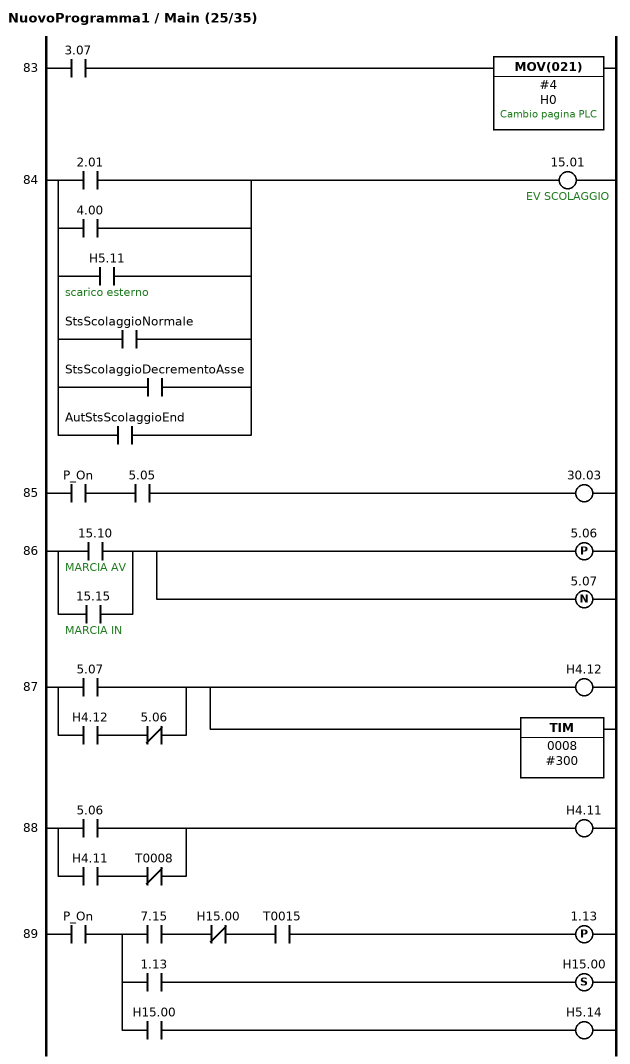
; [picture p24: NuovoProgramma1 / Main, rungs 83-89]
; rung 83
LD 3.07
MOV(021) #4 H0  ; Cambio pagina PLC
; rung 84
LD 2.01
OR 4.00
OR H5.11  ; scarico esterno
OR StsScolaggioNormale
OR StsScolaggioDecrementoAsse
OR AutStsScolaggioEnd
OUT 15.01  ; EV SCOLAGGIO
; rung 85
LD P_On
AND 5.05
OUT 30.03
; rung 86
LD 15.10  ; MARCIA AV
OR 15.15  ; MARCIA IN
DIFU(013) 5.06
DIFD(014) 5.07
; rung 87
LD 5.07
LD H4.12
ANDNOT 5.06
ORLD
OUT H4.12
TIM 0008 #300
; rung 88
LD 5.06
LD H4.11
ANDNOT T0008
ORLD
OUT H4.11
; rung 89
LD P_On
OUT TR0
AND 7.15
ANDNOT H15.00
AND T0015
DIFU(013) 1.13
LD TR0
AND 1.13
SET H15.00
LD TR0
AND H15.00
OUT H5.14

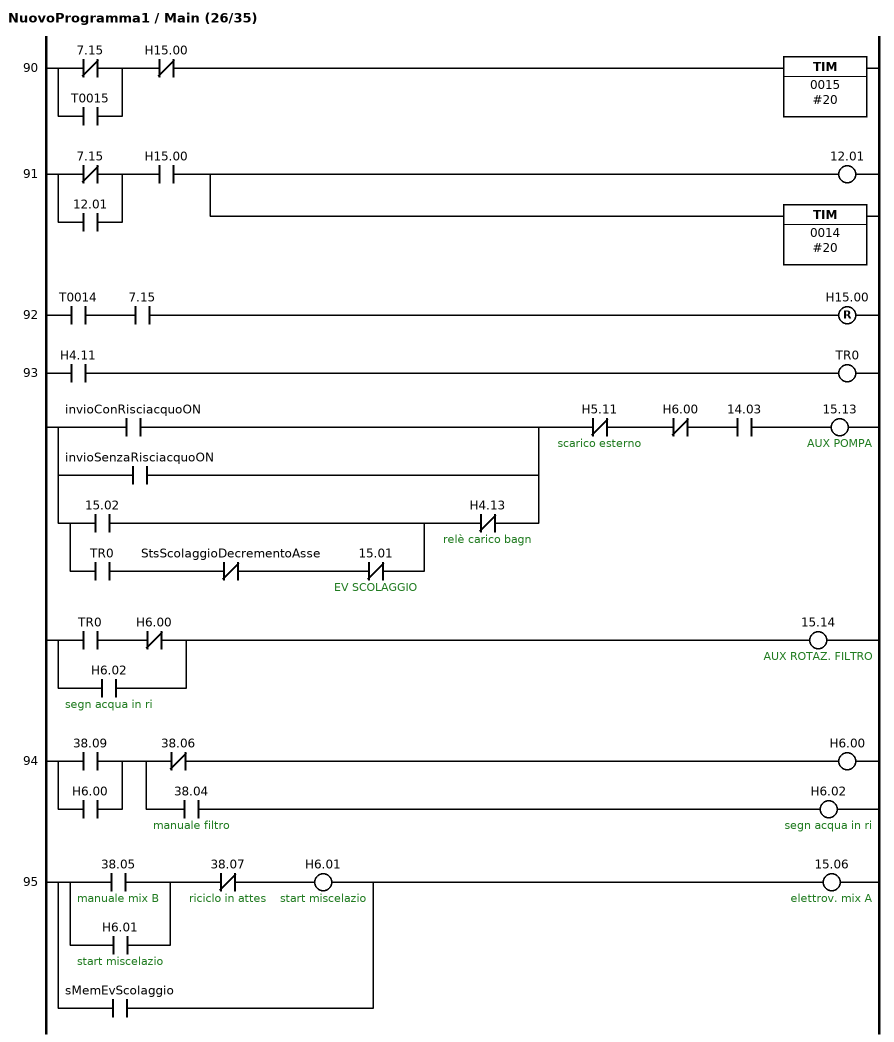
; rung 90
LDNOT 7.15
OR T0015
ANDNOT H15.00
TIM 0015 #20
; rung 91
LDNOT 7.15
OR 12.01
AND H15.00
OUT 12.01
TIM 0014 #20
; rung 92
LD T0014
AND 7.15
RSET H15.00
; rung 93
LD invioConRisciacquoON
OR invioSenzaRisciacquoON
LD 15.02
LD H4.11
OUT TR0
ANDNOT StsScolaggioDecrementoAsse
ANDNOT 15.01  ; EV SCOLAGGIO
ORLD
ANDNOT H4.13  ; relè carico bagn
ORLD
ANDNOT H5.11  ; scarico esterno
ANDNOT H6.00
AND 14.03
OUT 15.13  ; AUX POMPA
LD TR0
ANDNOT H6.00
OR H6.02  ; segn acqua in ri
OUT 15.14  ; AUX ROTAZ. FILTRO
; rung 94
LD 38.09
OR H6.00
OUT TR0
ANDNOT 38.06
OUT H6.00
LD TR0
AND 38.04  ; manuale filtro
OUT H6.02  ; segn acqua in ri
; rung 95
LD 38.05  ; manuale mix B
OR H6.01  ; start miscelazio
ANDNOT 38.07  ; riciclo in attes
OUT H6.01  ; start miscelazio
OR sMemEvScolaggio
OUT 15.06  ; elettrov. mix A

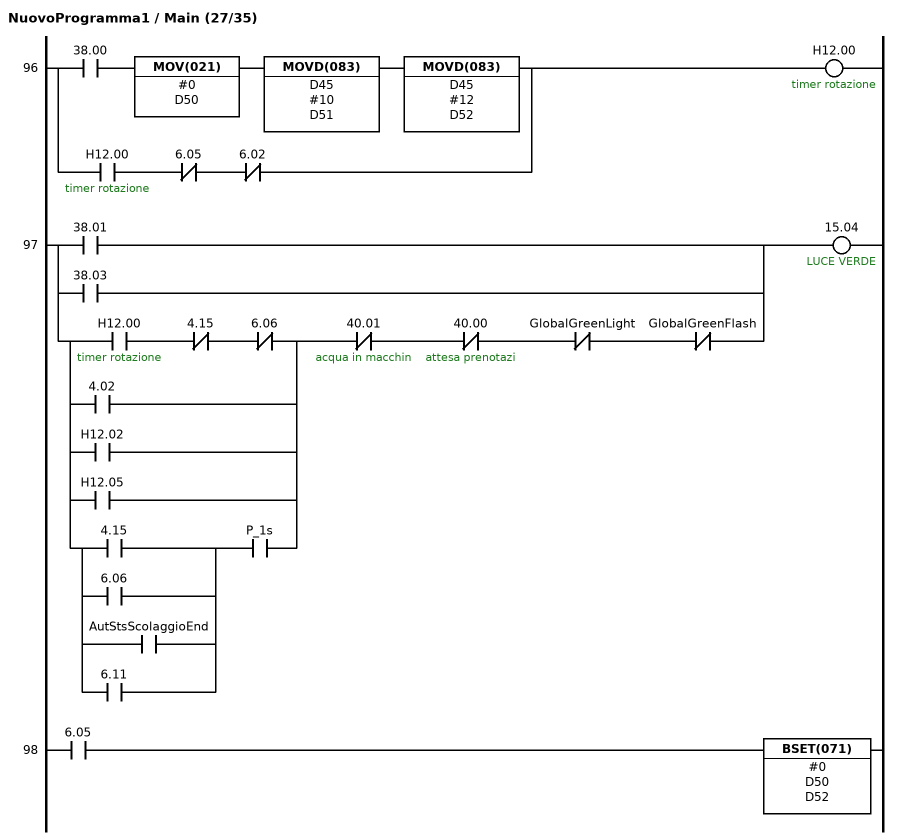
; rung 96
LD 38.00
MOV(021) #0 D50
MOVD(083) D45 #10 D51
MOVD(083) D45 #12 D52
LD H12.00  ; timer rotazione
ANDNOT 6.05
ANDNOT 6.02
ORLD
OUT H12.00  ; timer rotazione
; rung 97
LD 38.01
OR 38.03
LD H12.00  ; timer rotazione
ANDNOT 4.15
ANDNOT 6.06
OR 4.02
OR H12.02
OR H12.05
LD 4.15
OR 6.06
OR AutStsScolaggioEnd
OR 6.11
AND P_1s
ORLD
ANDNOT 40.01  ; acqua in macchin
ANDNOT 40.00  ; attesa prenotazi
ANDNOT GlobalGreenLight
ANDNOT GlobalGreenFlash
ORLD
OUT 15.04  ; LUCE VERDE
; rung 98
LD 6.05
BSET(071) #0 D50 D52

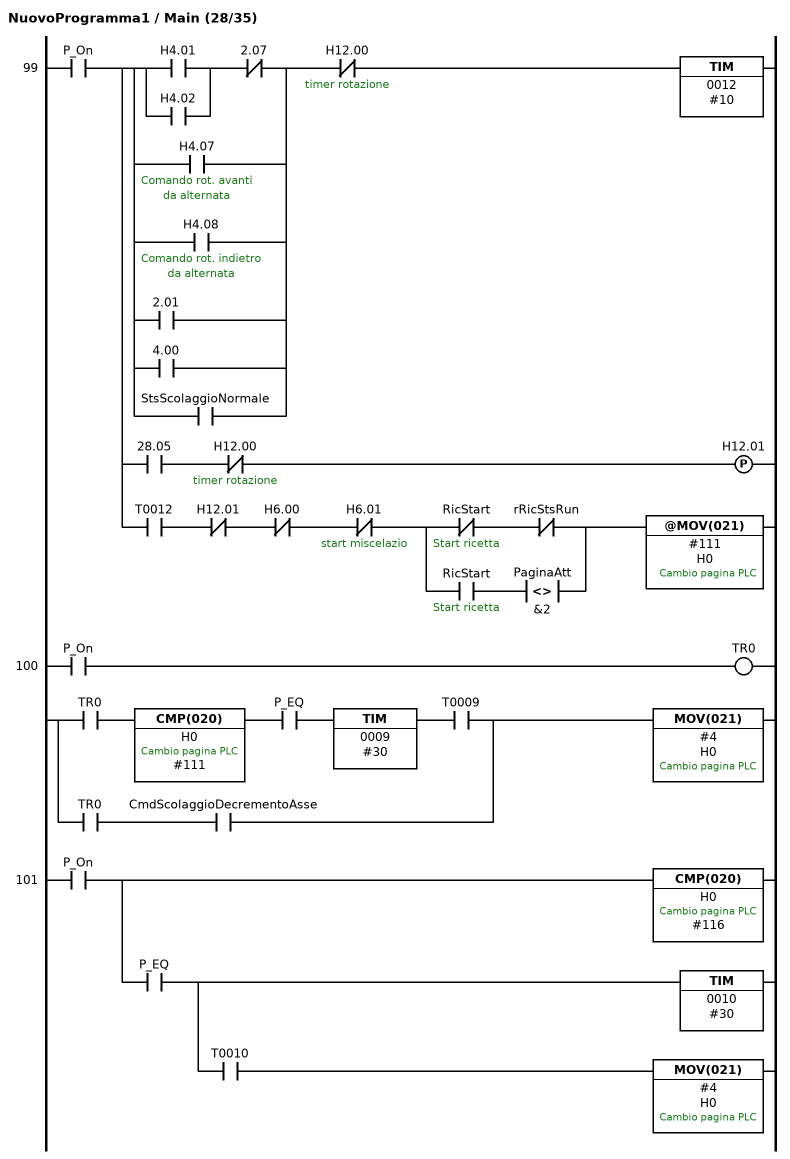
; rung 99
LD P_On
OUT TR0
LD H4.01
OR H4.02
ANDNOT 2.07
OR H4.07  ; Comando rot. avanti da alternata
OR H4.08  ; Comando rot. indietro da alternata
OR 2.01
OR 4.00
OR StsScolaggioNormale
ANDLD
ANDNOT H12.00  ; timer rotazione
TIM 0012 #10
LD TR0
AND 28.05
ANDNOT H12.00  ; timer rotazione
DIFU(013) H12.01
LD TR0
AND T0012
ANDNOT H12.01
ANDNOT H6.00
ANDNOT H6.01  ; start miscelazio
LDNOT RicStart  ; Start ricetta
ANDNOT rRicStsRun
LD RicStart  ; Start ricetta
AND<>(305) PaginaAtt &2
ORLD
ANDLD
@MOV(021) #111 H0  ; Cambio pagina PLC
; rung 100
LD P_On
OUT TR0
CMP(020) H0 #111  ; Cambio pagina PLC
AND P_EQ
TIM 0009 #30
AND T0009
LD TR0
AND CmdScolaggioDecrementoAsse
ORLD
MOV(021) #4 H0  ; Cambio pagina PLC
; rung 101
LD P_On
CMP(020) H0 #116  ; Cambio pagina PLC
AND P_EQ
TIM 0010 #30
AND T0010
MOV(021) #4 H0  ; Cambio pagina PLC

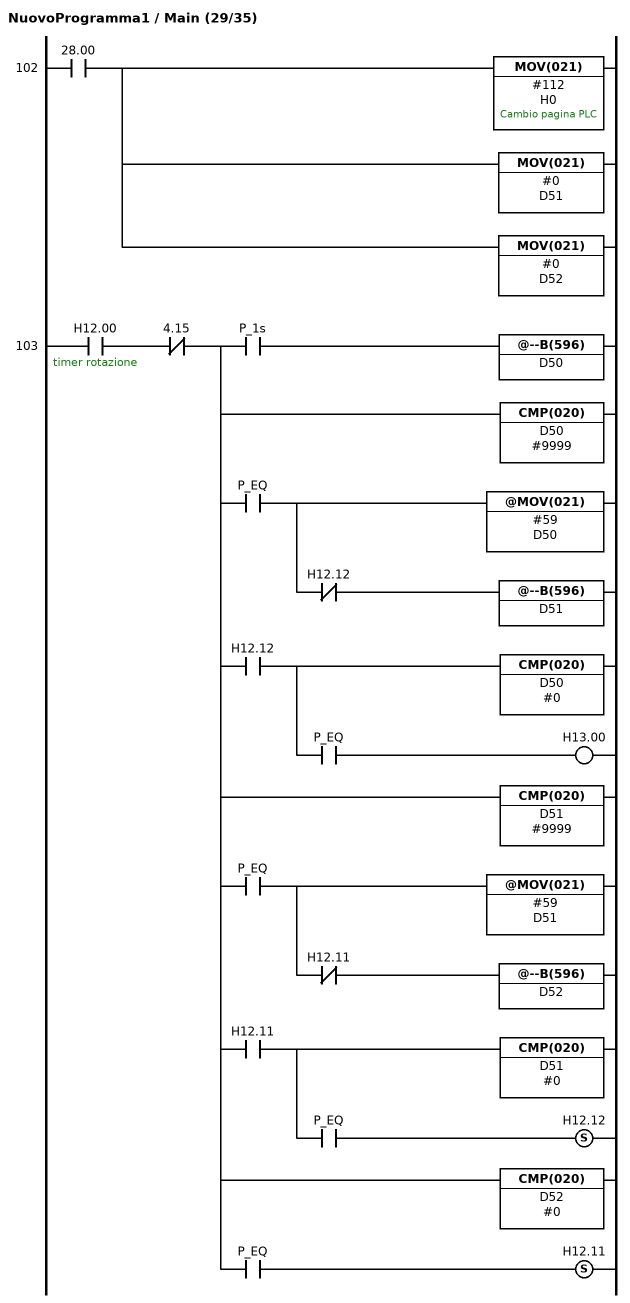
; rung 102
LD 28.00
MOV(021) #112 H0  ; Cambio pagina PLC
MOV(021) #0 D51
MOV(021) #0 D52
; rung 103
LD H12.00  ; timer rotazione
ANDNOT 4.15
OUT TR0
AND P_1s
@--B(596) D50
LD TR0
CMP(020) D50 #9999
AND P_EQ
@MOV(021) #59 D50
ANDNOT H12.12
@--B(596) D51
LD TR0
AND H12.12
CMP(020) D50 #0
AND P_EQ
OUT H13.00
LD TR0
CMP(020) D51 #9999
AND P_EQ
@MOV(021) #59 D51
ANDNOT H12.11
@--B(596) D52
LD TR0
AND H12.11
CMP(020) D51 #0
AND P_EQ
SET H12.12
LD TR0
CMP(020) D52 #0
AND P_EQ
SET H12.11

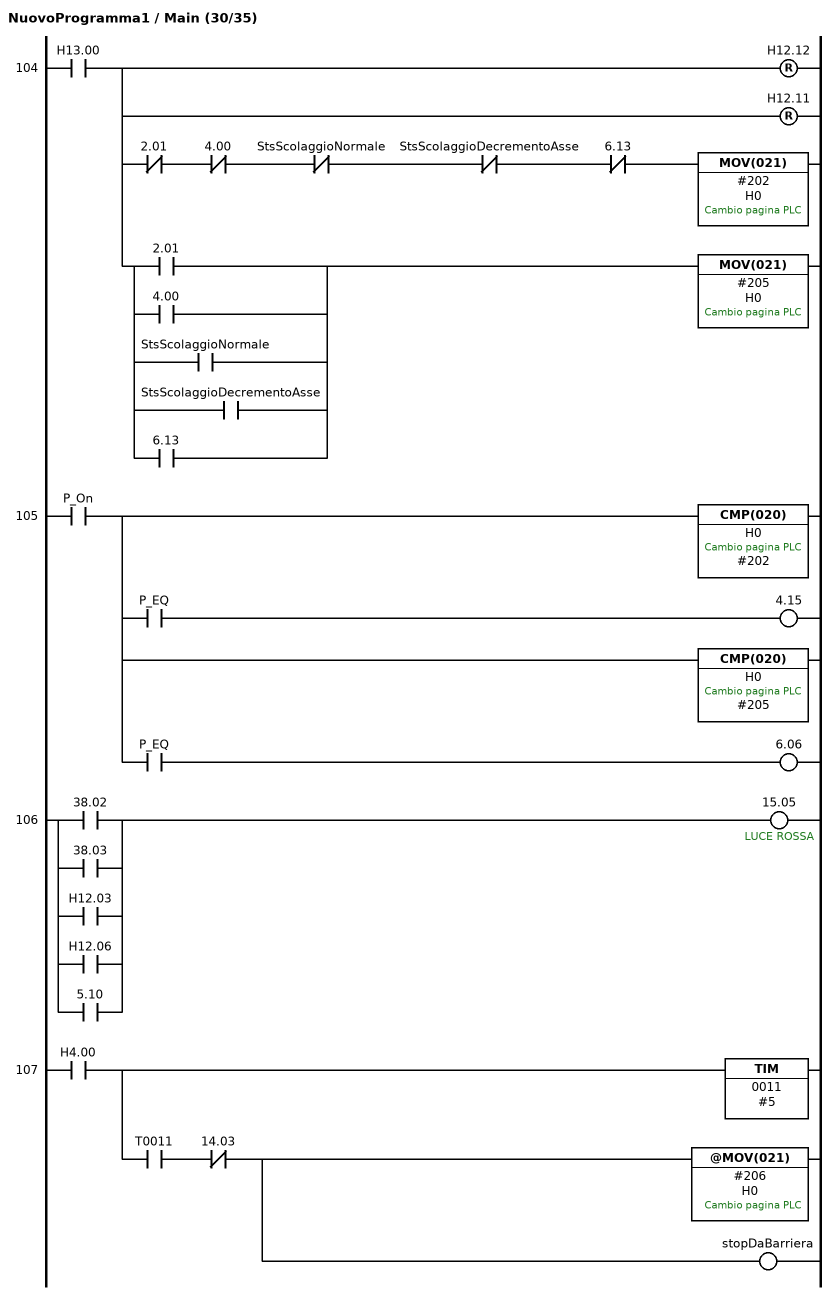
; rung 104
LD H13.00
OUT TR0
RSET H12.12
RSET H12.11
ANDNOT 2.01
ANDNOT 4.00
ANDNOT StsScolaggioNormale
ANDNOT StsScolaggioDecrementoAsse
ANDNOT 6.13
MOV(021) #202 H0  ; Cambio pagina PLC
LD TR0
LD 2.01
OR 4.00
OR StsScolaggioNormale
OR StsScolaggioDecrementoAsse
OR 6.13
ANDLD
MOV(021) #205 H0  ; Cambio pagina PLC
; rung 105
LD P_On
OUT TR0
CMP(020) H0 #202  ; Cambio pagina PLC
AND P_EQ
OUT 4.15
LD TR0
CMP(020) H0 #205  ; Cambio pagina PLC
AND P_EQ
OUT 6.06
; rung 106
LD 38.02
OR 38.03
OR H12.03
OR H12.06
OR 5.10
OUT 15.05  ; LUCE ROSSA
; rung 107
LD H4.00
TIM 0011 #5
AND T0011
ANDNOT 14.03
@MOV(021) #206 H0  ; Cambio pagina PLC
OUT stopDaBarriera

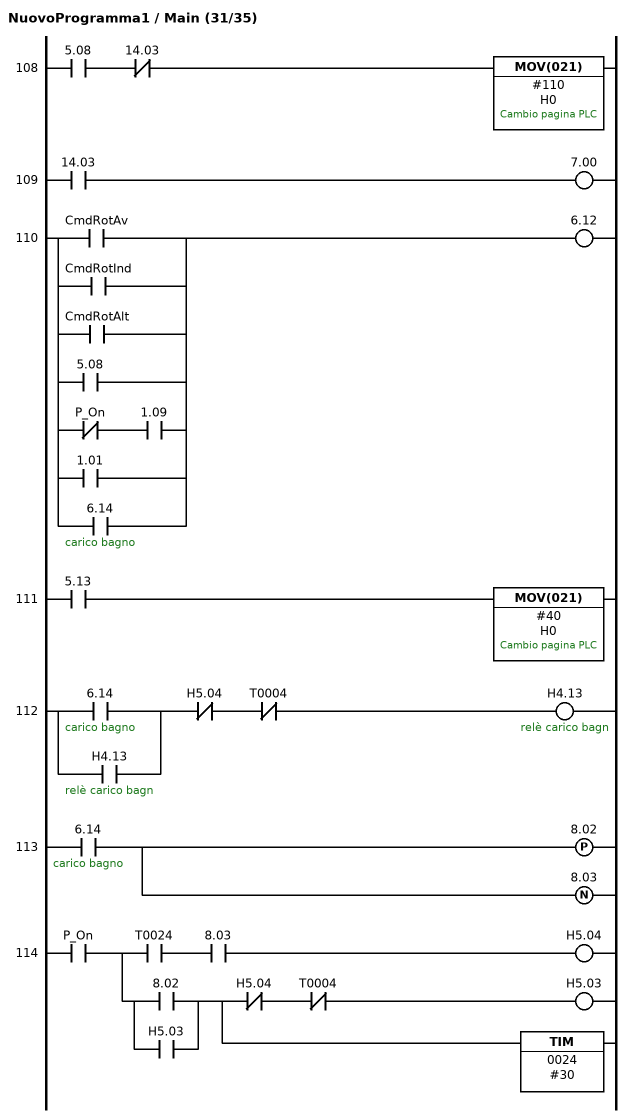
; rung 108
LD 5.08
ANDNOT 14.03
MOV(021) #110 H0  ; Cambio pagina PLC
; rung 109
LD 14.03
OUT 7.00
; rung 110
LD CmdRotAv
OR CmdRotInd
OR CmdRotAlt
OR 5.08
LDNOT P_On
AND 1.09
ORLD
OR 1.01
OR 6.14  ; carico bagno
OUT 6.12
; rung 111
LD 5.13
MOV(021) #40 H0  ; Cambio pagina PLC
; rung 112
LD 6.14  ; carico bagno
OR H4.13  ; relè carico bagn
ANDNOT H5.04
ANDNOT T0004
OUT H4.13  ; relè carico bagn
; rung 113
LD 6.14  ; carico bagno
DIFU(013) 8.02
DIFD(014) 8.03
; rung 114
LD P_On
OUT TR0
AND T0024
AND 8.03
OUT H5.04
LD TR0
LD 8.02
OR H5.03
ANDLD
OUT TR0
ANDNOT H5.04
ANDNOT T0004
OUT H5.03
LD TR0
TIM 0024 #30

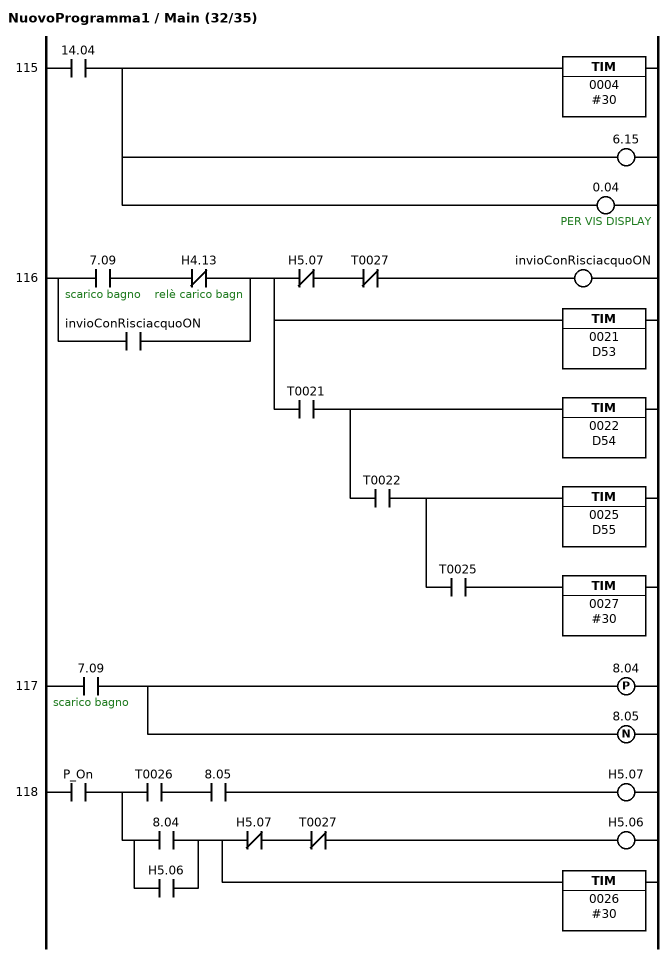
; rung 115
LD 14.04
TIM 0004 #30
OUT 6.15
OUT 0.04  ; PER VIS DISPLAY
; rung 116
LD 7.09  ; scarico bagno
ANDNOT H4.13  ; relè carico bagn
OR invioConRisciacquoON
OUT TR0
ANDNOT H5.07
ANDNOT T0027
OUT invioConRisciacquoON
LD TR0
TIM 0021 D53
AND T0021
TIM 0022 D54
AND T0022
TIM 0025 D55
AND T0025
TIM 0027 #30
; rung 117
LD 7.09  ; scarico bagno
DIFU(013) 8.04
DIFD(014) 8.05
; rung 118
LD P_On
OUT TR0
AND T0026
AND 8.05
OUT H5.07
LD TR0
LD 8.04
OR H5.06
ANDLD
OUT TR0
ANDNOT H5.07
ANDNOT T0027
OUT H5.06
LD TR0
TIM 0026 #30

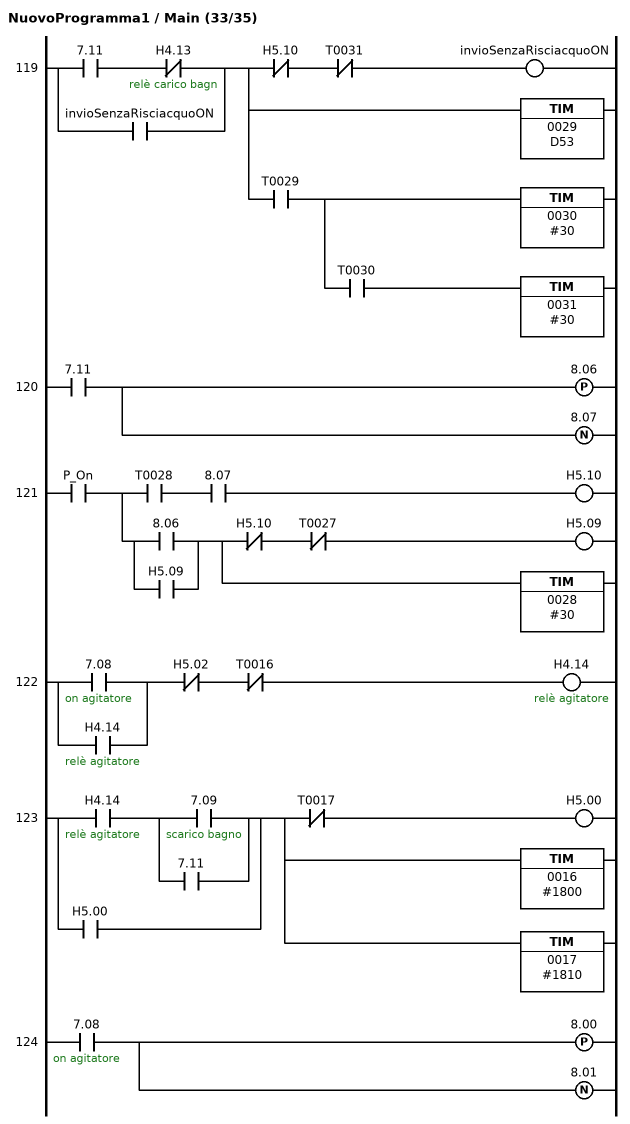
; rung 119
LD 7.11
ANDNOT H4.13  ; relè carico bagn
OR invioSenzaRisciacquoON
OUT TR0
ANDNOT H5.10
ANDNOT T0031
OUT invioSenzaRisciacquoON
LD TR0
TIM 0029 D53
AND T0029
TIM 0030 #30
AND T0030
TIM 0031 #30
; rung 120
LD 7.11
DIFU(013) 8.06
DIFD(014) 8.07
; rung 121
LD P_On
OUT TR0
AND T0028
AND 8.07
OUT H5.10
LD TR0
LD 8.06
OR H5.09
ANDLD
OUT TR0
ANDNOT H5.10
ANDNOT T0027
OUT H5.09
LD TR0
TIM 0028 #30
; rung 122
LD 7.08  ; on agitatore
OR H4.14  ; relè agitatore
ANDNOT H5.02
ANDNOT T0016
OUT H4.14  ; relè agitatore
; rung 123
LD H4.14  ; relè agitatore
LD 7.09  ; scarico bagno
OR 7.11
ANDLD
OR H5.00
OUT TR0
ANDNOT T0017
OUT H5.00
LD TR0
TIM 0016 #1800
TIM 0017 #1810
; rung 124
LD 7.08  ; on agitatore
DIFU(013) 8.00
DIFD(014) 8.01

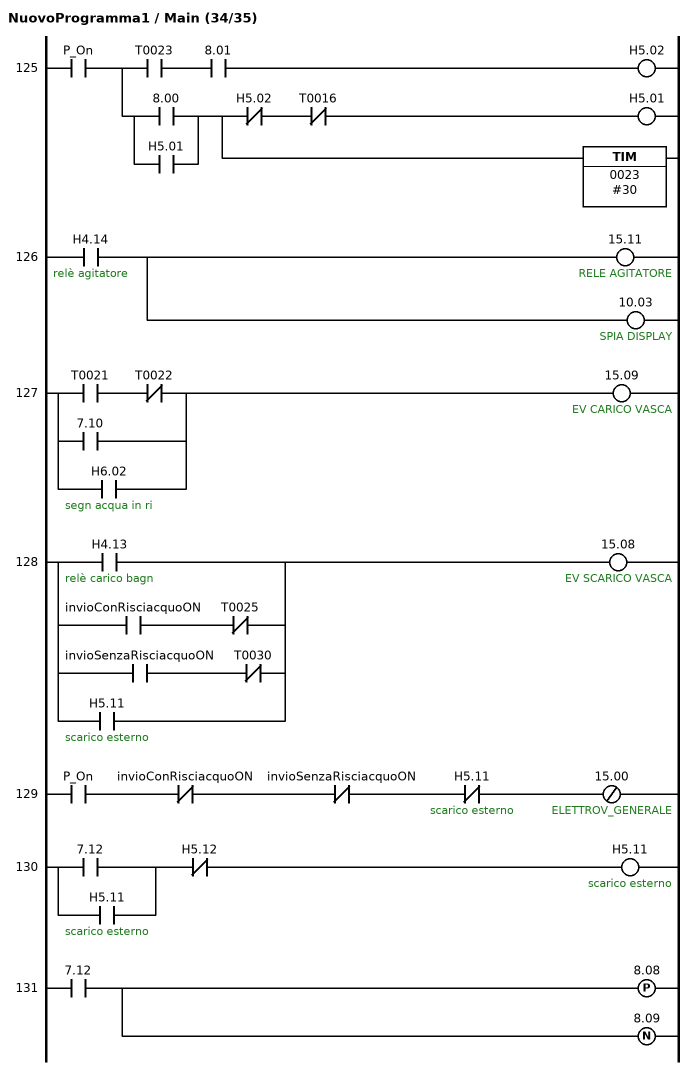
; rung 125
LD P_On
OUT TR0
AND T0023
AND 8.01
OUT H5.02
LD TR0
LD 8.00
OR H5.01
ANDLD
OUT TR0
ANDNOT H5.02
ANDNOT T0016
OUT H5.01
LD TR0
TIM 0023 #30
; rung 126
LD H4.14  ; relè agitatore
OUT 15.11  ; RELE AGITATORE
OUT 10.03  ; SPIA DISPLAY
; rung 127
LD T0021
ANDNOT T0022
OR 7.10
OR H6.02  ; segn acqua in ri
OUT 15.09  ; EV CARICO VASCA
; rung 128
LD H4.13  ; relè carico bagn
LD invioConRisciacquoON
ANDNOT T0025
ORLD
LD invioSenzaRisciacquoON
ANDNOT T0030
ORLD
OR H5.11  ; scarico esterno
OUT 15.08  ; EV SCARICO VASCA
; rung 129
LD P_On
ANDNOT invioConRisciacquoON
ANDNOT invioSenzaRisciacquoON
ANDNOT H5.11  ; scarico esterno
OUTNOT 15.00  ; ELETTROV_GENERALE
; rung 130
LD 7.12
OR H5.11  ; scarico esterno
ANDNOT H5.12
OUT H5.11  ; scarico esterno
; rung 131
LD 7.12
DIFU(013) 8.08
DIFD(014) 8.09

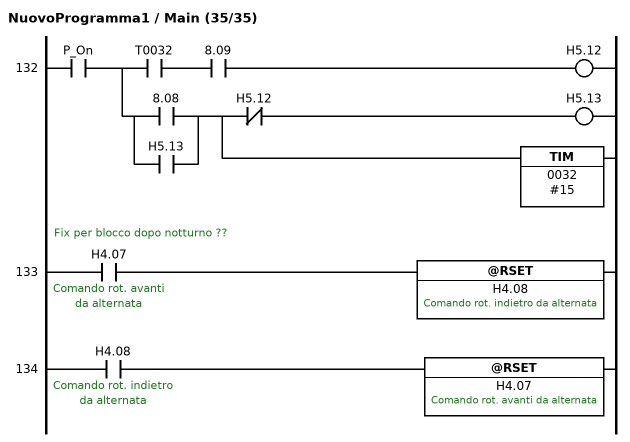
; rung 132
LD P_On
OUT TR0
AND T0032
AND 8.09
OUT H5.12
LD TR0
LD 8.08
OR H5.13
ANDLD
OUT TR0
ANDNOT H5.12
OUT H5.13
LD TR0
TIM 0032 #15
; rung 133: Fix per blocco dopo notturno ??
LD H4.07  ; Comando rot. avanti da alternata
@RSET H4.08  ; Comando rot. indietro da alternata
; rung 134
LD H4.08  ; Comando rot. indietro da alternata
@RSET H4.07  ; Comando rot. avanti da alternata

### Section GestioneLampeggianti

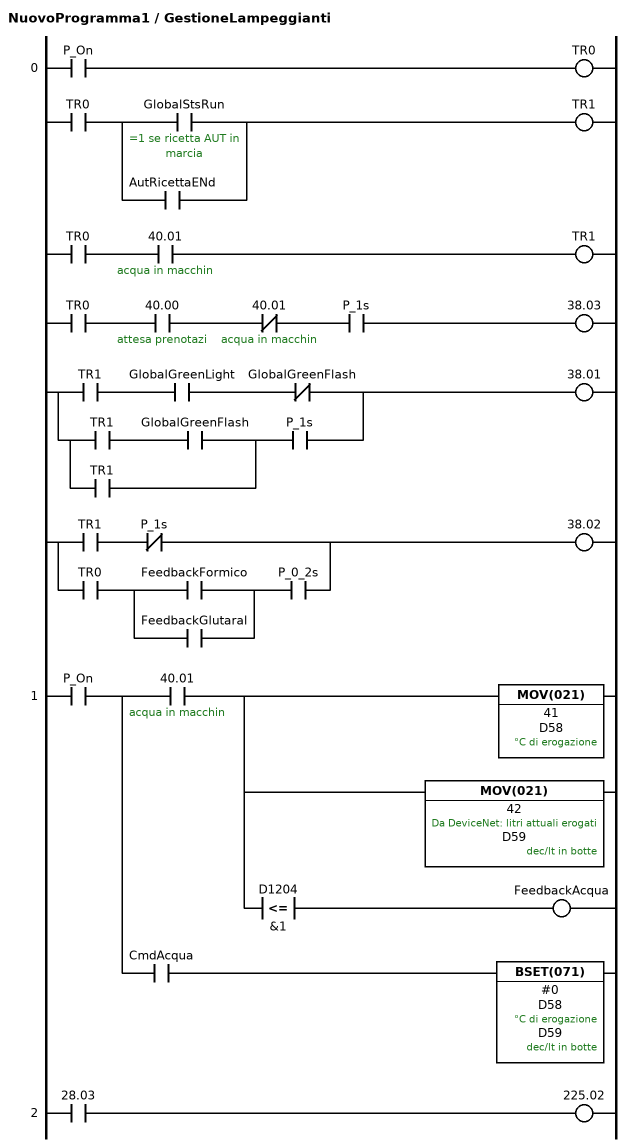
; rung 0
LD P_On
OUT TR0
AND 40.00  ; attesa prenotazi
ANDNOT 40.01  ; acqua in macchin
AND P_1s
OUT 38.03
LD TR0
LD GlobalStsRun  ; =1 se ricetta AUT in marcia
OR AutRicettaENd
ANDLD
OUT TR1
AND GlobalGreenLight
ANDNOT GlobalGreenFlash
LD TR1
AND GlobalGreenFlash
LD TR0
AND 40.01  ; acqua in macchin
OUT TR1
ORLD
AND P_1s
ORLD
OUT 38.01
LD TR1
ANDNOT P_1s
LD TR0
LD FeedbackFormico
OR FeedbackGlutaral
ANDLD
AND P_0_2s
ORLD
OUT 38.02
; rung 1
LD P_On
OUT TR0
AND 40.01  ; acqua in macchin
MOV(021) 41 D58  ; °C di erogazione
MOV(021) 42 D59  ; Da DeviceNet: litri attuali erogati, dec/lt in botte
AND<=(315) D1204 &1
OUT FeedbackAcqua
LD TR0
AND CmdAcqua
BSET(071) #0 D58 D59  ; °C di erogazione, dec/lt in botte
; rung 2
LD 28.03
OUT 225.02

### Section Sezione3

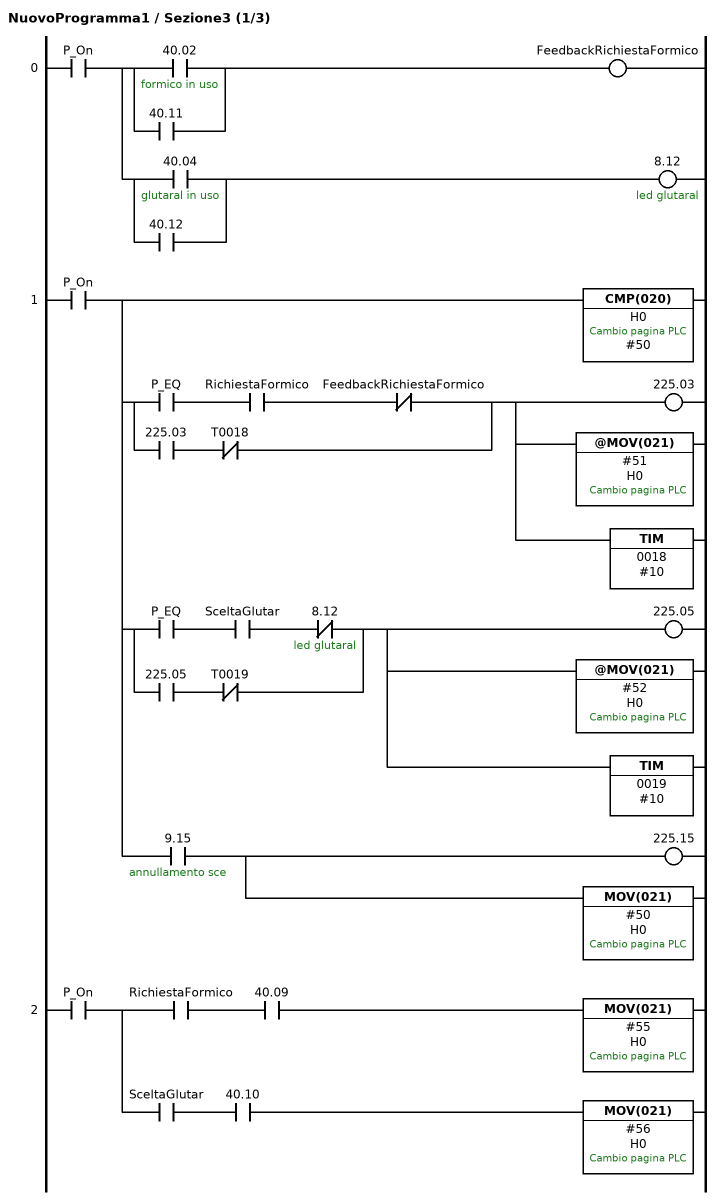
; rung 0
LD P_On
OUT TR0
LD 40.02  ; formico in uso
OR 40.11
ANDLD
OUT FeedbackRichiestaFormico
LD TR0
LD 40.04  ; glutaral in uso
OR 40.12
ANDLD
OUT 8.12  ; led glutaral
; rung 1
LD P_On
OUT TR0
CMP(020) H0 #50  ; Cambio pagina PLC
LD P_EQ
AND RichiestaFormico
ANDNOT FeedbackRichiestaFormico
LD 225.03
ANDNOT T0018
ORLD
ANDLD
OUT 225.03
@MOV(021) #51 H0  ; Cambio pagina PLC
TIM 0018 #10
LD TR0
LD P_EQ
AND SceltaGlutar
ANDNOT 8.12  ; led glutaral
LD 225.05
ANDNOT T0019
ORLD
ANDLD
OUT 225.05
@MOV(021) #52 H0  ; Cambio pagina PLC
TIM 0019 #10
LD TR0
AND 9.15  ; annullamento sce
OUT 225.15
MOV(021) #50 H0  ; Cambio pagina PLC
; rung 2
LD P_On
OUT TR0
AND RichiestaFormico
AND 40.09
MOV(021) #55 H0  ; Cambio pagina PLC
LD TR0
AND SceltaGlutar
AND 40.10
MOV(021) #56 H0  ; Cambio pagina PLC

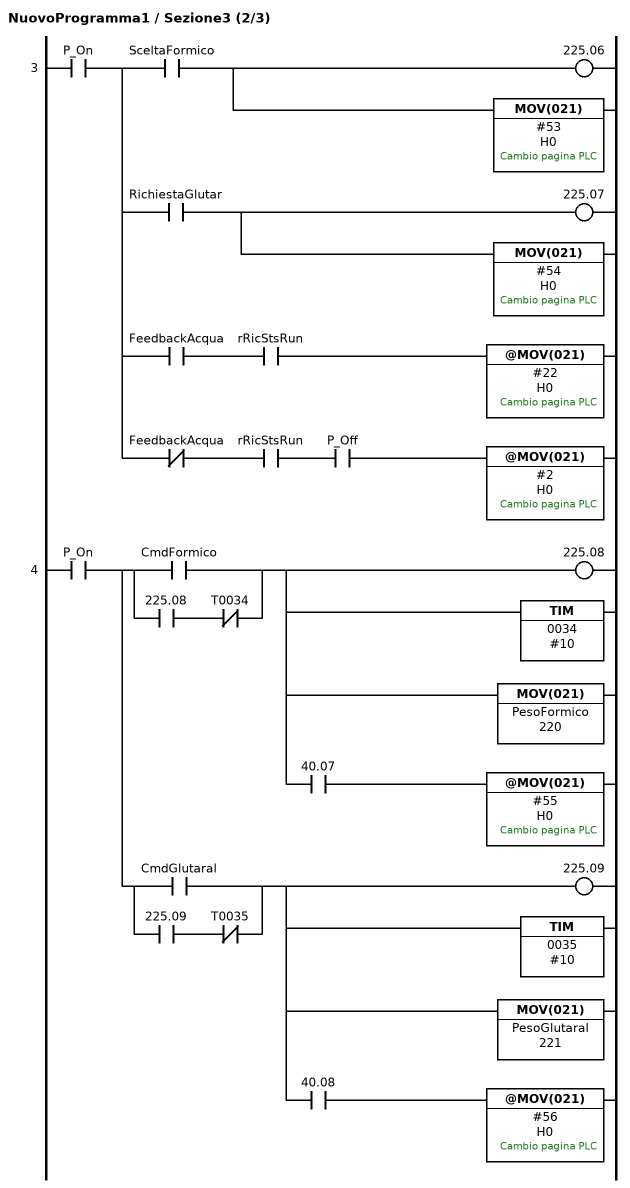
; rung 3
LD P_On
OUT TR0
AND SceltaFormico
OUT 225.06
MOV(021) #53 H0  ; Cambio pagina PLC
LD TR0
AND RichiestaGlutar
OUT 225.07
MOV(021) #54 H0  ; Cambio pagina PLC
LD TR0
AND FeedbackAcqua
AND rRicStsRun
@MOV(021) #22 H0  ; Cambio pagina PLC
LD TR0
ANDNOT FeedbackAcqua
AND rRicStsRun
AND P_Off
@MOV(021) #2 H0  ; Cambio pagina PLC
; rung 4
LD P_On
OUT TR0
LD CmdFormico
LD 225.08
ANDNOT T0034
ORLD
ANDLD
OUT 225.08
TIM 0034 #10
MOV(021) PesoFormico 220
AND 40.07
@MOV(021) #55 H0  ; Cambio pagina PLC
LD TR0
LD CmdGlutaral
LD 225.09
ANDNOT T0035
ORLD
ANDLD
OUT 225.09
TIM 0035 #10
MOV(021) PesoGlutaral 221
AND 40.08
@MOV(021) #56 H0  ; Cambio pagina PLC

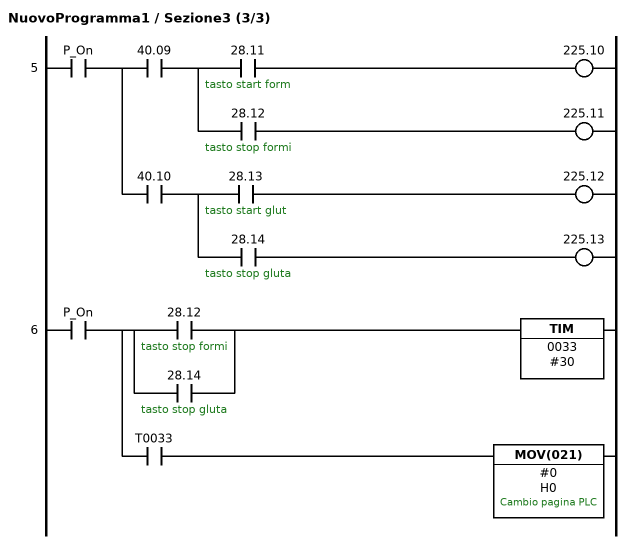
; rung 5
LD P_On
OUT TR0
AND 40.09
OUT TR1
AND 28.11  ; tasto start form
OUT 225.10
LD TR1
AND 28.12  ; tasto stop formi
OUT 225.11
LD TR0
AND 40.10
OUT TR0
AND 28.13  ; tasto start glut
OUT 225.12
LD TR0
AND 28.14  ; tasto stop gluta
OUT 225.13
; rung 6
LD P_On
OUT TR0
LD 28.12  ; tasto stop formi
OR 28.14  ; tasto stop gluta
ANDLD
TIM 0033 #30
LD TR0
AND T0033
MOV(021) #0 H0  ; Cambio pagina PLC
; rung 7
END(001)

## Program TaskRicette (cyclic task 1)
Local symbols
flagScansioniFallite BOOL
paginaAtt CHANNEL
ricStart BOOL
ricStsRun BOOL

### Section CambioPagina

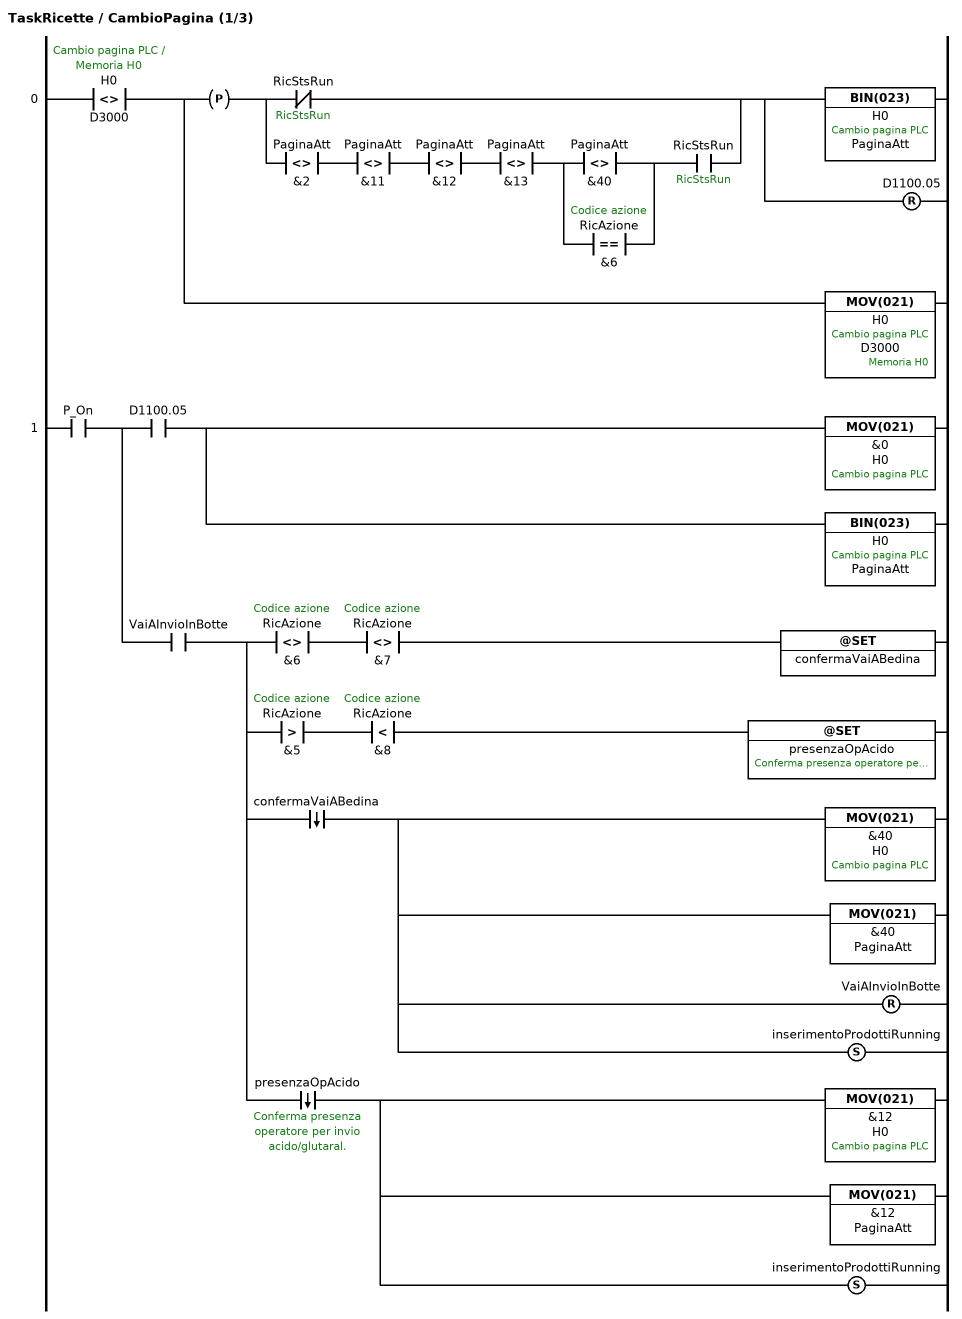
; rung 0
LD<>(305) H0 D3000  ; Cambio pagina PLC, Memoria H0
OUT TR0
UP(521)
LDNOT RicStsRun  ; RicStsRun
LD<>(305) PaginaAtt &2
AND<>(305) PaginaAtt &11
AND<>(305) PaginaAtt &12
AND<>(305) PaginaAtt &13
LD<>(305) PaginaAtt &40
OR=(300) RicAzione &6  ; Codice azione
ANDLD
AND RicStsRun  ; RicStsRun
ORLD
ANDLD
BIN(023) H0 PaginaAtt  ; Cambio pagina PLC
RSET D1100.05
LD TR0
MOV(021) H0 D3000  ; Cambio pagina PLC, Memoria H0
; rung 1
LD P_On
OUT TR0
AND D1100.05
MOV(021) &0 H0  ; Cambio pagina PLC
BIN(023) H0 PaginaAtt  ; Cambio pagina PLC
LD TR0
AND VaiAInvioInBotte
OUT TR0
AND<>(305) RicAzione &6  ; Codice azione
AND<>(305) RicAzione &7  ; Codice azione
@SET confermaVaiABedina
LD TR0
AND>(320) RicAzione &5  ; Codice azione
AND<(310) RicAzione &8  ; Codice azione
@SET presenzaOpAcido  ; Conferma presenza operatore per invio acido/glutaral.
LD TR0
%AND confermaVaiABedina
MOV(021) &40 H0  ; Cambio pagina PLC
MOV(021) &40 PaginaAtt
RSET VaiAInvioInBotte
SET inserimentoProdottiRunning
LD TR0
%AND presenzaOpAcido  ; Conferma presenza operatore per invio acido/glutaral.
MOV(021) &12 H0  ; Cambio pagina PLC
MOV(021) &12 PaginaAtt
SET inserimentoProdottiRunning

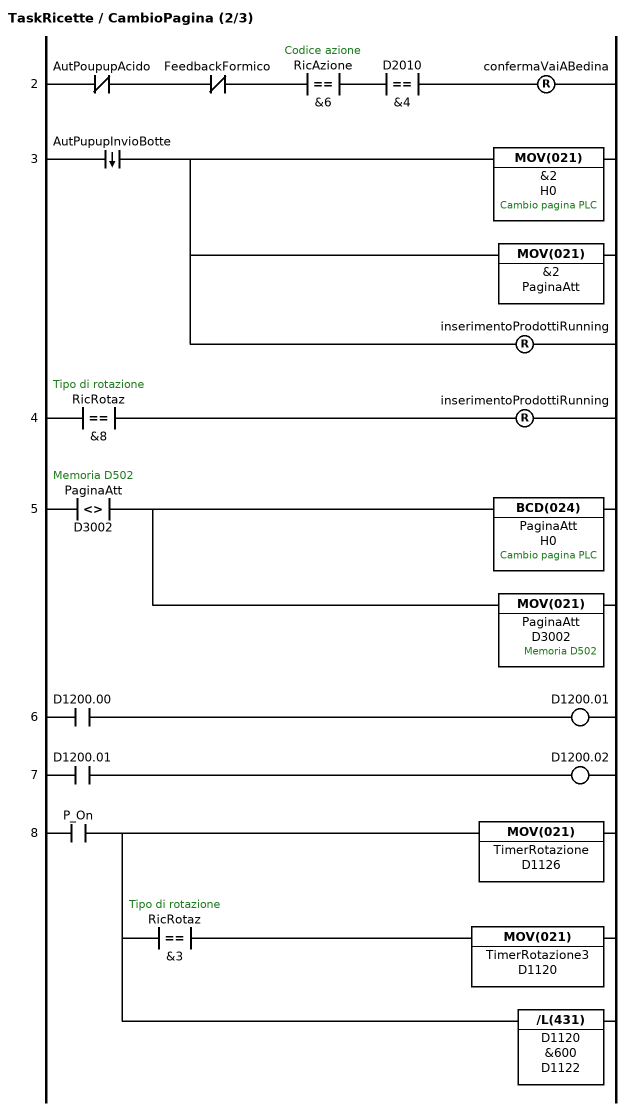
; rung 2
LDNOT AutPoupupAcido
ANDNOT FeedbackFormico
AND=(300) RicAzione &6  ; Codice azione
AND=(300) D2010 &4
RSET confermaVaiABedina
; rung 3
%LD AutPupupInvioBotte
MOV(021) &2 H0  ; Cambio pagina PLC
MOV(021) &2 PaginaAtt
RSET inserimentoProdottiRunning
; rung 4
LD=(300) RicRotaz &8  ; Tipo di rotazione
RSET inserimentoProdottiRunning
; rung 5
LD<>(305) PaginaAtt D3002  ; Memoria D502
BCD(024) PaginaAtt H0  ; Cambio pagina PLC
MOV(021) PaginaAtt D3002  ; Memoria D502
; rung 6
LD D1200.00
OUT D1200.01
; rung 7
LD D1200.01
OUT D1200.02
; rung 8
LD P_On
OUT TR0
MOV(021) TimerRotazione D1126
AND=(300) RicRotaz &3  ; Tipo di rotazione
MOV(021) TimerRotazione3 D1120
LD TR0
/L(431) D1120 &600 D1122

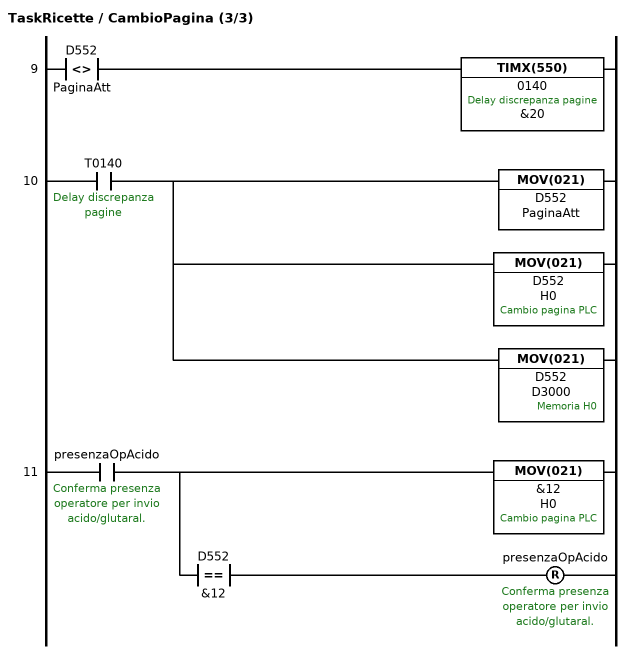
; rung 9
LD<>(305) D552 PaginaAtt
TIMX(550) 0140 &20  ; Delay discrepanza pagine
; rung 10
LD T0140  ; Delay discrepanza pagine
MOV(021) D552 PaginaAtt
MOV(021) D552 H0  ; Cambio pagina PLC
MOV(021) D552 D3000  ; Memoria H0
; rung 11
LD presenzaOpAcido  ; Conferma presenza operatore per invio acido/glutaral.
MOV(021) &12 H0  ; Cambio pagina PLC
AND=(300) D552 &12
RSET presenzaOpAcido  ; Conferma presenza operatore per invio acido/glutaral.

### Section Puntatori

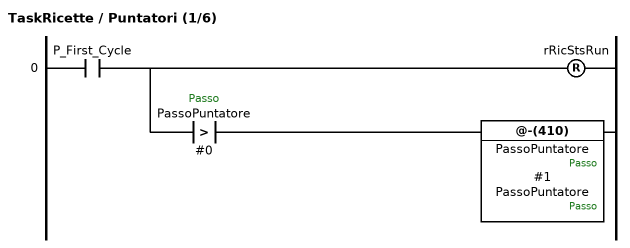
; rung 0
LD P_First_Cycle
RSET rRicStsRun
AND>(320) PassoPuntatore #0  ; Passo
@-(410) PassoPuntatore #1 PassoPuntatore  ; Passo

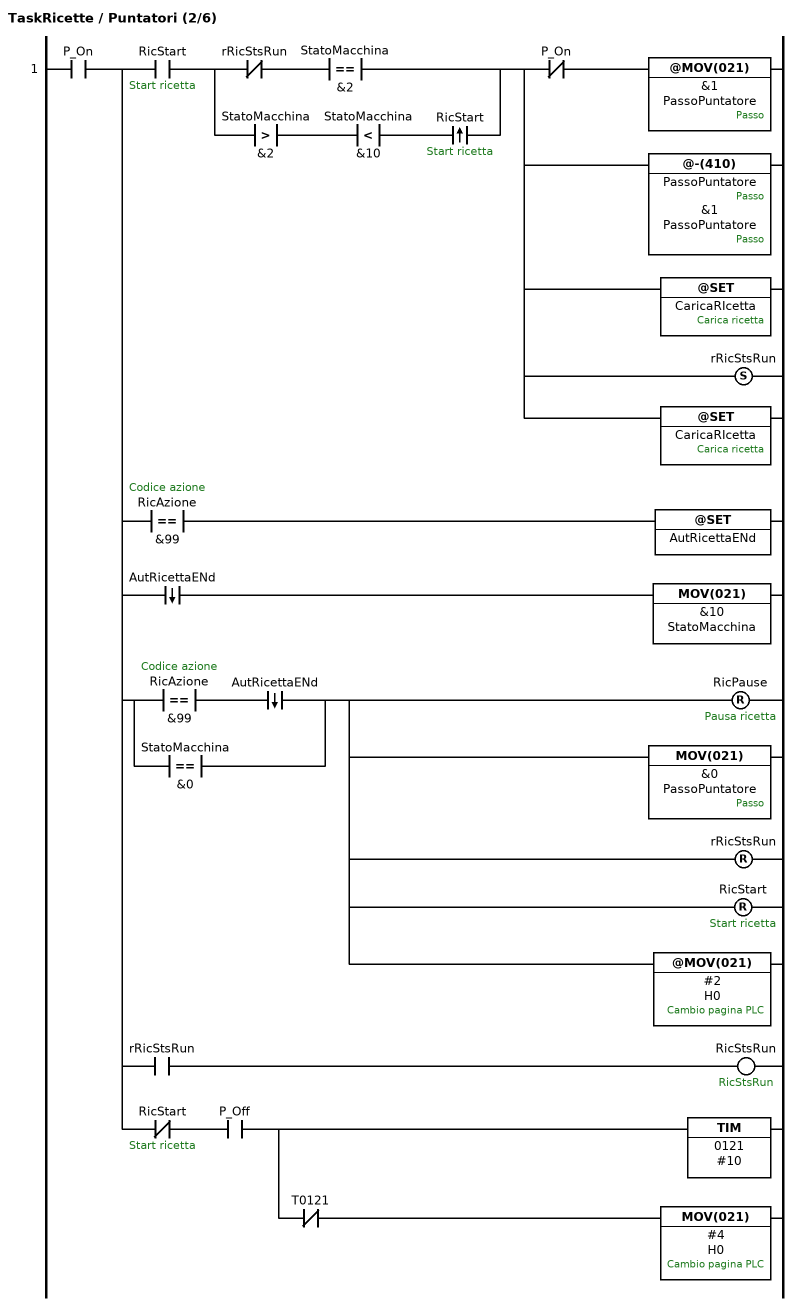
; rung 1
LD P_On
OUT TR0
AND RicStart  ; Start ricetta
LDNOT rRicStsRun
AND=(300) StatoMacchina &2
LD>(320) StatoMacchina &2
AND<(310) StatoMacchina &10
@AND RicStart  ; Start ricetta
ORLD
ANDLD
OUT TR1
ANDNOT P_On
@MOV(021) &1 PassoPuntatore  ; Passo
LD TR1
@-(410) PassoPuntatore &1 PassoPuntatore  ; Passo
@SET CaricaRIcetta  ; Carica ricetta
SET rRicStsRun
@SET CaricaRIcetta  ; Carica ricetta
LD TR0
AND=(300) RicAzione &99  ; Codice azione
@SET AutRicettaENd
LD TR0
%AND AutRicettaENd
MOV(021) &10 StatoMacchina
LD TR0
LD=(300) RicAzione &99  ; Codice azione
%AND AutRicettaENd
OR=(300) StatoMacchina &0
ANDLD
RSET RicPause  ; Pausa ricetta
MOV(021) &0 PassoPuntatore  ; Passo
RSET rRicStsRun
RSET RicStart  ; Start ricetta
@MOV(021) #2 H0  ; Cambio pagina PLC
LD TR0
AND rRicStsRun
OUT RicStsRun  ; RicStsRun
LD TR0
ANDNOT RicStart  ; Start ricetta
AND P_Off
TIM 0121 #10
ANDNOT T0121
MOV(021) #4 H0  ; Cambio pagina PLC

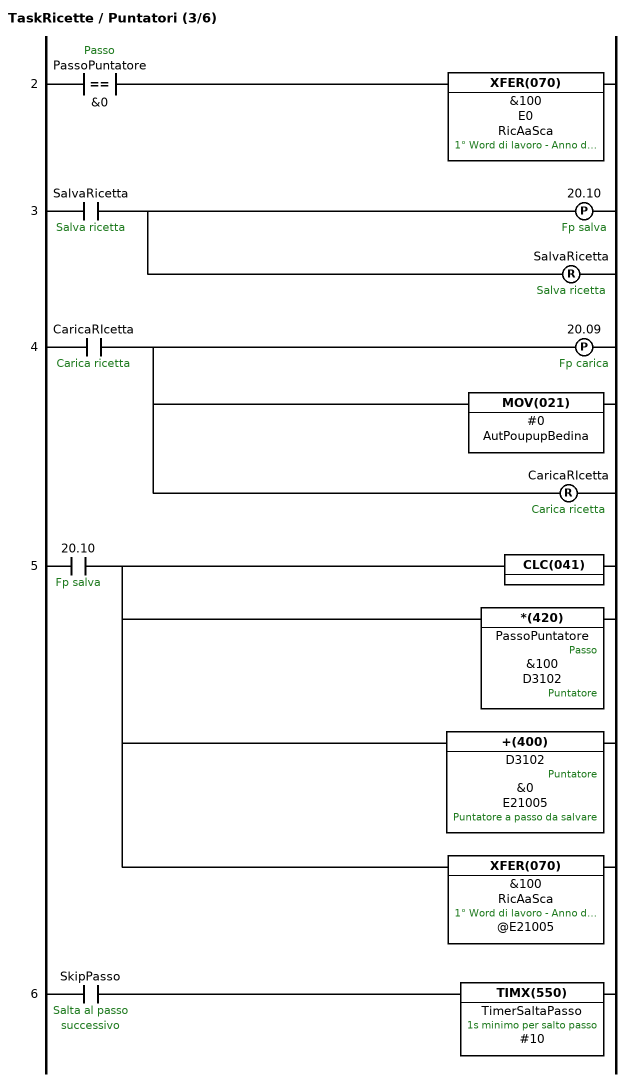
; rung 2
LD=(300) PassoPuntatore &0  ; Passo
XFER(070) &100 E0 RicAaSca  ; 1° Word di lavoro - Anno di produzione
; rung 3
LD SalvaRicetta  ; Salva ricetta
DIFU(013) 20.10  ; Fp salva
RSET SalvaRicetta  ; Salva ricetta
; rung 4
LD CaricaRIcetta  ; Carica ricetta
DIFU(013) 20.09  ; Fp carica
MOV(021) #0 AutPoupupBedina
RSET CaricaRIcetta  ; Carica ricetta
; rung 5
LD 20.10  ; Fp salva
CLC(041)
*(420) PassoPuntatore &100 D3102  ; Passo, Puntatore
+(400) D3102 &0 E21005  ; Puntatore, Puntatore a passo da salvare
XFER(070) &100 RicAaSca @E21005  ; 1° Word di lavoro - Anno di produzione
; rung 6
LD SkipPasso  ; Salta al passo successivo
TIMX(550) TimerSaltaPasso #10  ; 1s minimo per salto passo

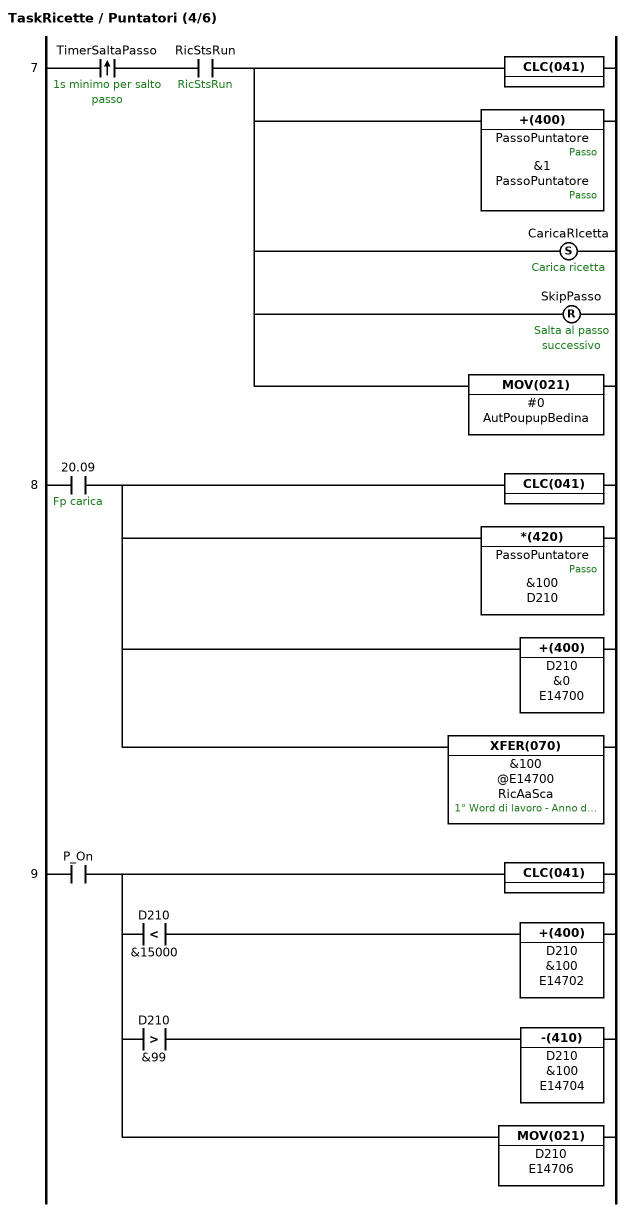
; rung 7
@LD TimerSaltaPasso  ; 1s minimo per salto passo
AND RicStsRun  ; RicStsRun
CLC(041)
+(400) PassoPuntatore &1 PassoPuntatore  ; Passo
SET CaricaRIcetta  ; Carica ricetta
RSET SkipPasso  ; Salta al passo successivo
MOV(021) #0 AutPoupupBedina
; rung 8
LD 20.09  ; Fp carica
CLC(041)
*(420) PassoPuntatore &100 D210  ; Passo
+(400) D210 &0 E14700
XFER(070) &100 @E14700 RicAaSca  ; 1° Word di lavoro - Anno di produzione
; rung 9
LD P_On
OUT TR0
CLC(041)
AND<(310) D210 &15000
+(400) D210 &100 E14702
LD TR0
AND>(320) D210 &99
-(410) D210 &100 E14704
LD TR0
MOV(021) D210 E14706

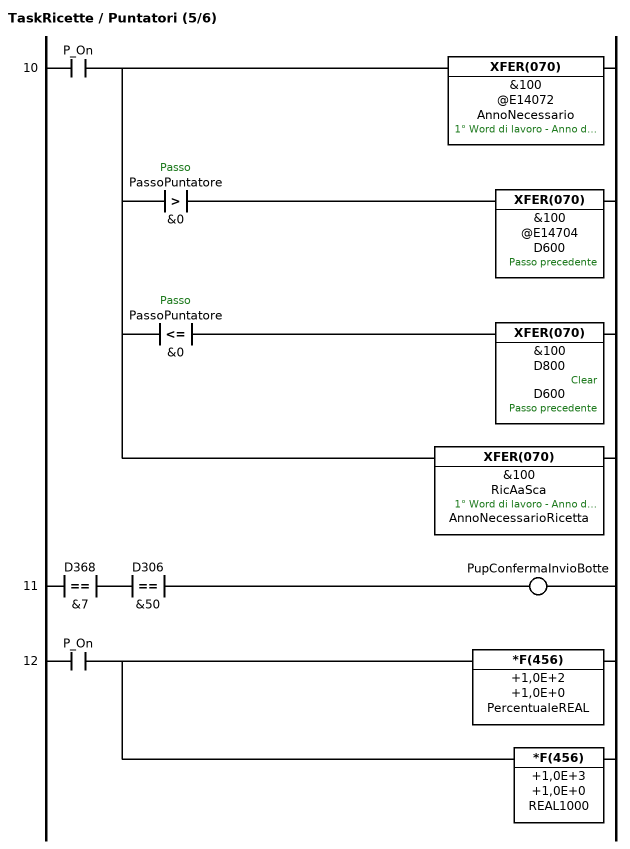
; rung 10
LD P_On
OUT TR0
XFER(070) &100 @E14072 AnnoNecessario  ; 1° Word di lavoro - Anno di produzione
AND>(320) PassoPuntatore &0  ; Passo
XFER(070) &100 @E14704 D600  ; Passo precedente
LD TR0
AND<=(315) PassoPuntatore &0  ; Passo
XFER(070) &100 D800 D600  ; Clear, Passo precedente
LD TR0
XFER(070) &100 RicAaSca AnnoNecessarioRicetta  ; 1° Word di lavoro - Anno di produzione
; rung 11
LD=(300) D368 &7
AND=(300) D306 &50
OUT PupConfermaInvioBotte
; rung 12
LD P_On
*F(456) +1,0E+2 +1,0E+0 PercentualeREAL
*F(456) +1,0E+3 +1,0E+0 REAL1000

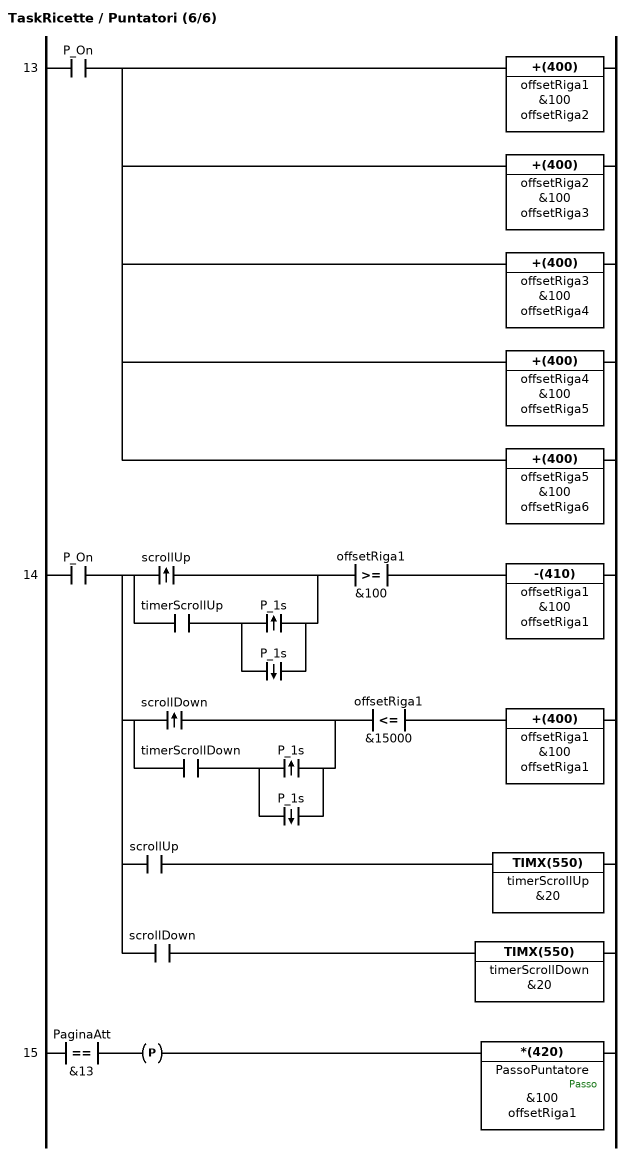
; rung 13
LD P_On
+(400) offsetRiga1 &100 offsetRiga2
+(400) offsetRiga2 &100 offsetRiga3
+(400) offsetRiga3 &100 offsetRiga4
+(400) offsetRiga4 &100 offsetRiga5
+(400) offsetRiga5 &100 offsetRiga6
; rung 14
LD P_On
OUT TR0
@LD scrollUp
LD timerScrollUp
@LD P_1s
%OR P_1s
ANDLD
ORLD
ANDLD
AND>=(325) offsetRiga1 &100
-(410) offsetRiga1 &100 offsetRiga1
LD TR0
@LD scrollDown
LD timerScrollDown
@LD P_1s
%OR P_1s
ANDLD
ORLD
ANDLD
AND<=(315) offsetRiga1 &15000
+(400) offsetRiga1 &100 offsetRiga1
LD TR0
AND scrollUp
TIMX(550) timerScrollUp &20
LD TR0
AND scrollDown
TIMX(550) timerScrollDown &20
; rung 15
LD=(300) PaginaAtt &13
UP(521)
*(420) PassoPuntatore &100 offsetRiga1  ; Passo

### Section StatoRicetta

